{attribute addProperty BoxType "EK1122-0000-0018"}
{attribute addProperty Id "Beckhoff_EJ2xxxsub_EK1100EK1100_179A0949162"}
{attribute addProperty CRC "2077021401"}
{attribute addProperty SizeInBites "16"}
{attribute addProperty SizeInBytes "2"}
TYPE Beckhoff_EJ2xxxEK1122_7BCCD4D9 EXTENDS EK1122_179A0949 :
STRUCT
	{attribute addProperty Name "Beckhoff_EJ2xxxsub_EK1100"}
	Beckhoff_EJ2xxxsub_EK1100 : EK1100_179A0949;
END_STRUCT
END_TYPE

(* stored: Version 1.2.0.0, ProductVersion 3.1.4024.9
   DUT Beckhoff_EJ2xxxEK1122_7BCCD4D9: Id {799aa5e6-3471-475a-8f1a-f62f0adbfa12} *)
